// TwinCAT 3 PLC project Utilities
// Title: Tc_Utilities
// Company: NewEngineer
// Author: https://github.com/phucpha
// ProjectVersion: 1.1.1.0
// Description: this is library use for Utilities for TC3.
// ProgramVersion: 3.1.4024.0
// libraries:
//   Tc2_Standard, * (Beckhoff Automation GmbH)
//   Tc2_System, * (Beckhoff Automation GmbH)
//   Tc2_Utilities, * (Beckhoff Automation GmbH)
//   Tc3_Module, * (Beckhoff Automation GmbH)
// project tree:
//   DUTs/ E_3rdPartyScadaWriteDataBase.TcDUT
//   DUTs/File Logger/ E_FileLoggerAddLogsState.TcDUT (not stored), E_FileLoggerInitState.TcDUT (not stored), E_FileLoggerSetNewPathState.TcDUT (not stored), E_FileLoggerState.TcDUT (not stored)
//   DUTs/Union/ U_Word2Dint.TcDUT, U_Word2Int.TcDUT (not stored), U_Word2Real.TcDUT
//   FC/ FUN_Compare_Timestructs.TcPOU, TimeStruct_To_sTimeAveva.TcPOU
//   FC/StringMerge/ FUN_MergeLongStrings10.TcPOU, FUN_MergeStrings10.TcPOU, FUN_MergeStrings3.TcPOU, FUN_MergeStrings4.TcPOU (not stored), FUN_MergeStrings5.TcPOU, FUN_MergeStrings6.TcPOU
//   FC/Systemtime to String/ FUN_TimestructToDate.TcPOU, FUN_TimestructToTime.TcPOU
//   FC/ValueToTime/ F_lrMinute2Time.TcPOU, F_LrSecond2Time.TcPOU (not stored), F_Time2lrHour.TcPOU, F_Time2lrMinute.TcPOU (not stored), F_Time2lrSecond.TcPOU
//   GVLs/ GVL.TcGVL
//   / PlcTask.TcTTO
//   POUs/0_Checks/Checks/ CheckBounds.TcPOU, CheckDivDInt.TcPOU, CheckDivLInt.TcPOU, CheckDivLReal.TcPOU, CheckDivReal.TcPOU, CheckPointer.TcPOU, CheckRangeSigned.TcPOU, CheckRangeUnsigned.TcPOU, P_Checks.TcPOU
//   POUs/0_Checks/ GVL_Checks.TcGVL
//   POUs/Alarms/ FB_Alarm.TcPOU, I_Alarm.TcIO
//   POUs/CrossCheckTime/ FB_TimeCrossCheck2System.TcPOU
//   POUs/FileLogger/ FB_FileLogger.TcPOU (not stored), I_FileLogger.TcIO (not stored)
//   Version/ Global_Version.TcGVL
// real-time tasks:
//   TASK PlcTask: cycle T#10ms, priority 20, ADS port 350

CONFIGURATION Utilities
    RESOURCE PLC ON TwinCAT3
        TASK PlcTask(INTERVAL := T#10ms, PRIORITY := 20);
    END_RESOURCE
END_CONFIGURATION

// ---- DUTs/E_3rdPartyScadaWriteDataBase.TcDUT
{attribute 'strict'}
TYPE E_3rdPartyScadaWriteDataBase :
(
	DATABASE_WRITE_WAIT_START := 0,
	DATABASE_WRITE_PREPARE_VALUE, 
	DATABASE_WRITE_SEND_REQUEST,
	DATABASE_WRITE_WAIT_RESPONSE
	
);
END_TYPE

// ---- DUTs/Union/U_Word2Dint.TcDUT
TYPE U_Word2Dint :
UNION
	iWord	: ARRAY[0..1] OF WORD;
	idInt	: DINT;
END_UNION
END_TYPE

// ---- DUTs/Union/U_Word2Real.TcDUT
TYPE U_Word2Real :
UNION
	iWord: ARRAY [0..1] OF WORD;
	rReal: REAL;
END_UNION
END_TYPE

// ---- GVLs/GVL.TcGVL
VAR_GLOBAL
	fbMachineTime : FB_LocalSystemTime;
	fbMachineLogger : FB_FileLogger;
END_VAR

// ---- POUs/0_Checks/GVL_Checks.TcGVL
{attribute 'qualified_only'}
VAR_GLOBAL PERSISTENT
	dCheckBounds					: DINT;			// Licznik przekroczen zakresu indexow, np. tablic
	dCheckDivDInt					: DINT;			// Licznik prob dzielenia Dint przez 0
	dCheckDivLInt					: DINT; 		// Licznik prob dzielenia LInt przez 0
	dCheckDivLReal					: DINT; 		// Licznik prob dzielenia LREAL przez 0
	dCheckDivReal					: DINT; 		// Licznik prob dzielenia REAL przez 0
	dCheckRangeSigned				: DINT;			// Licznik przekroczen liczby znakowej
	dCheckRangeUnsigned				: DINT; 		// Licznik przekroczen liczby bezznakowej
END_VAR

// ---- Version/Global_Version.TcGVL
{attribute 'TcGenerated'}
{attribute 'no-analysis'}
{attribute 'linkalways'}
// This function has been automatically generated from the project information.
VAR_GLOBAL CONSTANT
	{attribute 'const_non_replaced'}
	stLibVersion_Tc_Utilities : ST_LibVersion := (iMajor := 1, iMinor := 1, iBuild := 1, iRevision := 0, nFlags := 0, sVersion := '1.1.1.0');
END_VAR

// ---- POUs/Alarms/I_Alarm.TcIO
INTERFACE I_Alarm

PROPERTY AlarmNumber : UINT
GET
END_GET
SET
END_SET
END_PROPERTY

PROPERTY Description : String
GET
END_GET
SET
END_SET
END_PROPERTY

METHOD Get : BOOL
VAR_INPUT
END_VAR
VAR_OUTPUT

END_VAR
END_METHOD

METHOD Reset : BOOL
VAR_INPUT
END_VAR
END_METHOD

METHOD Set : BOOL
VAR
END_VAR
VAR_INPUT
	bIn	:	BOOL;
END_VAR
END_METHOD

PROPERTY TimeOfOccur : TIMESTRUCT
GET
END_GET
END_PROPERTY

END_INTERFACE

// ---- FC/FUN_Compare_Timestructs.TcPOU
FUNCTION FUN_Compare_Timestructs : SINT //returns: 1 IF ts1 is older, -1 if ts2 is older, 0 if equal
VAR_INPUT
	ts1	:	TIMESTRUCT;
	ts2	:	TIMESTRUCT;
END_VAR
VAR
END_VAR

//OUTPUT: 1 IF ts1 is older, -1 if ts2 is older, 0 if equal
IF (ts1.wYear=ts2.wYear) THEN
	IF (ts1.wMonth=ts2.wMonth) THEN
		IF (ts1.wDay=ts2.wDay) THEN
			IF (ts1.wHour=ts2.wHour) THEN
				IF (ts1.wMinute=ts2.wMinute) THEN
					IF (ts1.wSecond=ts2.wSecond) THEN
						IF (ts1.wMilliseconds=ts2.wMilliseconds) THEN
							FUN_Compare_Timestructs:=0;
						ELSIF (ts1.wMilliseconds>ts2.wMilliseconds) THEN
								FUN_Compare_Timestructs:=-1;
						ELSE
								FUN_Compare_Timestructs:=1;
						END_IF
						
					ELSIF (ts1.wSecond>ts2.wSecond) THEN
						FUN_Compare_Timestructs:=-1;
					ELSE
						FUN_Compare_Timestructs:=1;
					END_IF
					
				ELSIF (ts1.wMinute>ts2.wMinute) THEN
					FUN_Compare_Timestructs:=-1;
				ELSE
					FUN_Compare_Timestructs:=1;
				END_IF
				
			ELSIF (ts1.wHour>ts2.wHour) THEN
				FUN_Compare_Timestructs:=-1;
			ELSE
				FUN_Compare_Timestructs:=1;
			END_IF
		
		ELSIF (ts1.wDay>ts2.wDay) THEN
			FUN_Compare_Timestructs:=-1;
		ELSE
			FUN_Compare_Timestructs:=1;
		END_IF
	
	ELSIF (ts1.wMonth>ts2.wMonth) THEN
		FUN_Compare_Timestructs:=-1;
	ELSE
		FUN_Compare_Timestructs:=1;
	END_IF
	
ELSIF (ts1.wYear>ts2.wYear) THEN
	FUN_Compare_Timestructs:=-1;
ELSE
	FUN_Compare_Timestructs:=1;
END_IF

END_FUNCTION

// ---- FC/StringMerge/FUN_MergeLongStrings10.TcPOU
(* 
:Description: This function is used to merge 10 long strings
*)
FUNCTION FUN_MergeLongStrings10 : STRING(2000)
VAR_INPUT
	sStr1	: STRING(2000);
	sStr2	: STRING(2000);
	sStr3	: STRING(2000);
	sStr4	: STRING(2000);
	sStr5	: STRING(2000);
	sStr6	: STRING(2000);
	sStr7	: STRING(2000);
	sStr8	: STRING(2000);
	sStr9	: STRING(2000);
	sStr10	: STRING(2000);
END_VAR
VAR
	sStrTemp1 :	STRING(2000);
	sStrTemp2 :	STRING(2000);
END_VAR

CONCAT2(ADR(sStr1),ADR(sStr2),ADR(sStrTemp1),SIZEOF(sStrTemp1));
CONCAT2(ADR(sStrTemp1),ADR(sStr3),ADR(sStrTemp2),SIZEOF(sStrTemp2));
CONCAT2(ADR(sStrTemp2),ADR(sStr4),ADR(sStrTemp1),SIZEOF(sStrTemp1));
CONCAT2(ADR(sStrTemp1),ADR(sStr5),ADR(sStrTemp2),SIZEOF(sStrTemp2));
CONCAT2(ADR(sStrTemp2),ADR(sStr6),ADR(sStrTemp1),SIZEOF(sStrTemp1));
CONCAT2(ADR(sStrTemp1),ADR(sStr7),ADR(sStrTemp2),SIZEOF(sStrTemp2));
CONCAT2(ADR(sStrTemp2),ADR(sStr8),ADR(sStrTemp1),SIZEOF(sStrTemp1));
CONCAT2(ADR(sStrTemp1),ADR(sStr9),ADR(sStrTemp2),SIZEOF(sStrTemp2));
CONCAT2(ADR(sStrTemp2),ADR(sStr10),ADR(FUN_MergeLongStrings10),SIZEOF(FUN_MergeLongStrings10));

END_FUNCTION

// ---- FC/StringMerge/FUN_MergeStrings10.TcPOU
(* 
:Description: This function is used to merge 10 strings
*)
FUNCTION FUN_MergeStrings10 : STRING
VAR_INPUT
	sStr1	: STRING;		(* First string in merge row *)
	sStr2	: STRING;		(* Second string in merge row *)
	sStr3	: STRING;		(* Third string in merge row *)
	sStr4	: STRING(500);	(* Fourth string in merge row *)
	sStr5	: STRING(500);	(* Fifth string in merge row *)
	sStr6	: STRING(500);	(* Sixth string in merge row *)
	sStr7	: STRING(500);	(* Seventh string in merge row *)
	sStr8	: STRING;		(* Eight string in merge row *)
	sStr9	: STRING;		(* Ninth string in merge row *)
	sStr10	: STRING;		(* Tenth string in merge row *)
END_VAR

FUN_MergeStrings10 := CONCAT(sStr1,sStr2);
FUN_MergeStrings10 := CONCAT(FUN_MergeStrings10,sStr3);
FUN_MergeStrings10 := CONCAT(FUN_MergeStrings10,sStr4);
FUN_MergeStrings10 := CONCAT(FUN_MergeStrings10,sStr5);
FUN_MergeStrings10 := CONCAT(FUN_MergeStrings10,sStr6);
FUN_MergeStrings10 := CONCAT(FUN_MergeStrings10,sStr7);
FUN_MergeStrings10 := CONCAT(FUN_MergeStrings10,sStr8);
FUN_MergeStrings10 := CONCAT(FUN_MergeStrings10,sStr9);
FUN_MergeStrings10 := CONCAT(FUN_MergeStrings10,sStr10);

END_FUNCTION

// ---- FC/StringMerge/FUN_MergeStrings3.TcPOU
(* 
:Description: This function is used to merge 5 strings
*)
FUNCTION FUN_MergeStrings3 : STRING
VAR_INPUT
	sStr1	: STRING;			(* Fifth string in merge row *)
	sStr2	: STRING;			(* Fourth string in merge row *)
	sStr3	: STRING;			(* Fourth string in merge row *)

END_VAR

FUN_MergeStrings3 := CONCAT(sStr1,sStr2);
FUN_MergeStrings3 := CONCAT(FUN_MergeStrings3,sStr3);

END_FUNCTION

// ---- FC/StringMerge/FUN_MergeStrings5.TcPOU
(* 
:Description: This function is used to merge 5 strings
*)
FUNCTION FUN_MergeStrings5 : STRING
VAR_INPUT
	sStr1	: STRING;		(* First string in merge row *)
	sStr2	: STRING;		(* Second string in merge row *)
	sStr3	: STRING;		(* Third string in merge row *)
	sStr4	: STRING;		(* Fourth string in merge row *)
	sStr5	: STRING;		(* Fifth string in merge row *)

END_VAR

FUN_MergeStrings5 := CONCAT(sStr1,sStr2);
FUN_MergeStrings5 := CONCAT(FUN_MergeStrings5, sStr3);
FUN_MergeStrings5 := CONCAT(FUN_MergeStrings5, sStr4);
FUN_MergeStrings5 := CONCAT(FUN_MergeStrings5, sStr5);

END_FUNCTION

// ---- FC/StringMerge/FUN_MergeStrings6.TcPOU
(* 
:Description: This function is used to merge 6 strings
*)
FUNCTION FUN_MergeStrings6 : STRING(300)
VAR_INPUT
	sStr1	: STRING;		(* First string in merge row *)
	sStr2	: STRING;		(* Second string in merge row *)
	sStr3	: STRING;		(* Third string in merge row *)
	sStr4	: STRING;		(* Fourth string in merge row *)
	sStr5	: STRING;		(* Fifth string in merge row *)
	sStr6	: STRING;		(* Sixth string in merge row *)
END_VAR

FUN_MergeStrings6 := CONCAT(sStr1,sStr2);
FUN_MergeStrings6 := CONCAT(FUN_MergeStrings6, sStr3);
FUN_MergeStrings6 := CONCAT(FUN_MergeStrings6, sStr4);
FUN_MergeStrings6 := CONCAT(FUN_MergeStrings6, sStr5);
FUN_MergeStrings6 := CONCAT(FUN_MergeStrings6, sStr6);

END_FUNCTION

// ---- FC/Systemtime to String/FUN_TimestructToDate.TcPOU
FUNCTION FUN_TimestructToDate : STRING
VAR_INPUT
	stTime : TIMESTRUCT;
END_VAR
VAR
	sTime : STRING;
END_VAR

sTime := SYSTEMTIME_TO_STRING(stTime);
FUN_TimestructToDate := LEFT(sTime,10);

END_FUNCTION

// ---- FC/Systemtime to String/FUN_TimestructToTime.TcPOU
FUNCTION FUN_TimestructToTime : STRING
VAR_INPUT
	stTime : TIMESTRUCT;
END_VAR
VAR
	sTime : STRING;
END_VAR

sTime := SYSTEMTIME_TO_STRING(stTime);
FUN_TimestructToTime := RIGHT(sTime,12);

END_FUNCTION

// ---- FC/TimeStruct_To_sTimeAveva.TcPOU
FUNCTION TimeStruct_To_sTimeAveva : STRING// convert TIMESTRUCT TO MONTH/DAY/YEAR HOUR:MINUTE: SECOND ( FORMAT 'MM/DD/YYYY HH:MM:SS' )
VAR_INPUT
	timestruct 	: TIMESTRUCT;
	typeFormat	: UINT := 0; (* 	0: 'MM/DD/YYYY HH:MM:SS'
									1: 'MMDDYYYY'
									2: 'YYYYMMDD'
									3: 'DDMMYYYY'
									4: 'YYYY-MM-DD HH:MM:SS' 
									5: 'YYYY-MM-DD HH:MM:SS.XXX'
													*)
	
END_VAR
VAR
	sYear : STRING;
	sMonth : STRING;
	sDay : STRING;
	sHour : STRING;
	sMinute : STRING;
	sSecond : STRING;
	sMilisecond	: STRING;
	concate1 : STRING;
	
END_VAR

	sYear := WORD_TO_STRING(timestruct.wYear);
	sMonth := WORD_TO_STRING(timestruct.wMonth);
	sDay 	:= WORD_TO_STRING(timestruct.wDay);
	
	sHour := WORD_TO_STRING(timestruct.wHour);
	sMinute := WORD_TO_STRING(timestruct.wMinute);
	sSecond 	:= WORD_TO_STRING(timestruct.wSecond);
	sMilisecond := WORD_TO_STRING(timestruct.wMilliseconds);
	
	IF timestruct.wMonth <10 THEN
		sMonth := CONCAT('0', smonth);
	END_IF
	
	IF timestruct.wDay <10 THEN
		sDay := CONCAT('0', sday);
	END_IF
	
	IF timestruct.wHour <10 THEN
		sHour := CONCAT('0', shour);
	END_IF
	IF timestruct.wSecond <10 THEN
		ssecond := CONCAT('0', ssecond);
	END_IF
	IF timestruct.wMinute <10 THEN
		sMinute := CONCAT('0', sminute);
	END_IF
	
	IF timestruct.wMilliseconds < 10  THEN
		sMilisecond :=  CONCAT('00', sMilisecond);
	ELSIF timestruct.wMilliseconds < 100 THEN
		sMilisecond :=  CONCAT('0', sMilisecond);
	END_IF
	
CASE typeFormat OF
	0://0: 'MM/DD/YYYY HH:MM:SS'
		concate1 := CONCAT( smonth, '/');
		concate1 := CONCAT( concate1, sDay);
		concate1 := CONCAT( concate1, '/');
		concate1 := CONCAT( concate1, sYear);
		concate1 := CONCAT( concate1, ' ');
		concate1 := CONCAT( concate1, shour);
		concate1 := CONCAT( concate1, ':');
		concate1 := CONCAT( concate1, sminute);
		concate1 := CONCAT( concate1, ':');
		concate1 := CONCAT( concate1, ssecond);
	
	1: //1: 'MMDDYYYY'
		concate1 := CONCAT( smonth, sDay);
		concate1 := CONCAT( concate1, sYear);
		
	2: 	//2: 'YYYYMMDD'
		concate1 := CONCAT( syear, smonth);
		concate1 := CONCAT( concate1, sday);	
		
	3: 	//3: 'DDMMYYYY'
		concate1 := CONCAT( sday, smonth);
		concate1 := CONCAT( concate1, syear);	
	4: //'YYYY-MM-DD HH:MM:SS' 
		concate1 := CONCAT( syear, '-');//YYYY-
		concate1 := CONCAT ( concate1, smonth);//YYYY-MM
		concate1 := CONCAT( concate1, '-');//YYYY-MM-
		concate1 := CONCAT( concate1, SDAY);//YYYY-MM-DD
		concate1 := CONCAT( concate1, ' ');//'YYYY-MM-DD '
		concate1 := CONCAT( concate1, shour);//'YYYY-MM-DD HH
		concate1 := CONCAT( concate1, ':');//'YYYY-MM-DD HH:
		concate1 := CONCAT( concate1, sminute);//'YYYY-MM-DD HH:MM
		concate1 := CONCAT( concate1, ':');//'YYYY-MM-DD HH:MM:
		concate1 := CONCAT( concate1, ssecond);//'YYYY-MM-DD HH:MM:SS
	5: (*need addition code*)
		concate1 := CONCAT( syear, '-');//YYYY-
		concate1 := CONCAT ( concate1, smonth);//YYYY-MM
		concate1 := CONCAT( concate1, '-');//YYYY-MM-
		concate1 := CONCAT( concate1, SDAY);//YYYY-MM-DD
		concate1 := CONCAT( concate1, ' ');//'YYYY-MM-DD '
		concate1 := CONCAT( concate1, shour);//'YYYY-MM-DD HH
		concate1 := CONCAT( concate1, ':');//'YYYY-MM-DD HH:
		concate1 := CONCAT( concate1, sminute);//'YYYY-MM-DD HH:MM
		concate1 := CONCAT( concate1, ':');//'YYYY-MM-DD HH:MM:
		concate1 := CONCAT( concate1, ssecond);//'YYYY-MM-DD HH:MM:SS
		concate1 := CONCAT( concate1, '.');//'YYYY-MM-DD HH:MM:SS.
		concate1 := CONCAT( concate1, sMilisecond); ////'YYYY-MM-DD HH:MM:SS.xxx
		
	ELSE
		concate1 := '';
END_CASE

TimeStruct_To_sTimeAveva := concate1;

END_FUNCTION

// ---- FC/ValueToTime/F_lrMinute2Time.TcPOU
FUNCTION F_lrMinute2Time : Time
VAR_INPUT
	lrMinute	: lreal;
END_VAR
VAR
END_VAR

F_lrMinute2Time := LREAL_TO_TIME( lrMinute*60*1000);

END_FUNCTION

// ---- FC/ValueToTime/F_Time2lrHour.TcPOU
FUNCTION F_Time2lrHour : lreal
VAR_INPUT
	t : TIME;
END_VAR

VAR
END_VAR

F_Time2lrHour := time_to_lreal(t)*2.777777777777777*expt(10,-7); // *0.001*0.01666666667 = /1000/60/60

END_FUNCTION

// ---- FC/ValueToTime/F_Time2lrSecond.TcPOU
FUNCTION F_Time2lrSecond : lreal
VAR_INPUT
	t : TIME;
END_VAR
VAR
END_VAR

F_Time2lrSecond := time_to_lreal(t)/1000;

END_FUNCTION

// ---- POUs/0_Checks/Checks/CheckBounds.TcPOU
// Implicitly generated code : DO NOT EDIT
FUNCTION CheckBounds : DINT
VAR_INPUT
	index, lower, upper: DINT;
END_VAR

// Implicitly generated code : Only an Implementation suggestion
IF  index < lower THEN
	CheckBounds := lower;
	GVL_Checks.dCheckBounds := GVL_Checks.dCheckBounds + 1;
//	ADSLOGSTR(4,'Checks critical error - index out of range','');
ELSIF  index > upper THEN
	CheckBounds := upper;
	GVL_Checks.dCheckBounds := GVL_Checks.dCheckBounds + 1;
//	ADSLOGSTR(4,'Checks critical error - index out of range','');
ELSE  
	CheckBounds := index;
END_IF

END_FUNCTION

// ---- POUs/0_Checks/Checks/CheckDivDInt.TcPOU
// Implicitly generated code : DO NOT EDIT
FUNCTION CheckDivDInt : DINT
VAR_INPUT
	divisor:DINT;
END_VAR

// Implicitly generated code : Only an Implementation suggestion
IF divisor = 0 THEN
	CheckDivDInt:=1;
	GVL_Checks.dCheckDivDInt := GVL_Checks.dCheckDivDInt + 1;
	ADSLOGSTR(4,'Checks critical error - DINT variable divided by 0.','');
ELSE
	CheckDivDInt:=divisor;
END_IF

END_FUNCTION

// ---- POUs/0_Checks/Checks/CheckDivLInt.TcPOU
// Implicitly generated code : DO NOT EDIT
FUNCTION CheckDivLInt : LINT
VAR_INPUT
	divisor:LINT;
END_VAR

// Implicitly generated code : Only an Implementation suggestion
IF divisor = 0 THEN
	CheckDivLInt:=1;
	GVL_Checks.dCheckDivLInt := GVL_Checks.dCheckDivLInt + 1;
	ADSLOGSTR(4,'Checks critical error - LINT variable divided by 0.','');
ELSE
	CheckDivLInt:=divisor;
END_IF

END_FUNCTION

// ---- POUs/0_Checks/Checks/CheckDivLReal.TcPOU
// Implicitly generated code : DO NOT EDIT
FUNCTION CheckDivLReal : LREAL
VAR_INPUT
	divisor:LREAL;
END_VAR

// Implicitly generated code : Only an Implementation suggestion
IF divisor = 0 THEN
	CheckDivLReal:=1;
	GVL_Checks.dCheckDivLReal := GVL_Checks.dCheckDivLReal + 1;
	ADSLOGSTR(4,'Checks critical error - DINT variable divided by 0.','');
ELSE
	CheckDivLReal:=divisor;
END_IF

END_FUNCTION

// ---- POUs/0_Checks/Checks/CheckDivReal.TcPOU
// Implicitly generated code : DO NOT EDIT
FUNCTION CheckDivReal : REAL
VAR_INPUT
	divisor:REAL;
END_VAR

// Implicitly generated code : Only an Implementation suggestion
IF divisor = 0 THEN
	CheckDivReal:=1;
	GVL_Checks.dCheckDivReal := GVL_Checks.dCheckDivReal + 1;
	ADSLOGSTR(4,'Checks critical error - DINT variable divided by 0.','');
ELSE
	CheckDivReal:=divisor;
END_IF

END_FUNCTION

// ---- POUs/0_Checks/Checks/CheckPointer.TcPOU
// Implicitly generated code : DO NOT EDIT
FUNCTION CheckPointer : POINTER TO BYTE
VAR_INPUT 
	ptToTest : POINTER TO BYTE; // Destination address of the pointer
	iSize : DINT;		        // Size of the type the pointer points to. (e.g: 20 for POINTER TO ARRAY [0..9] OF INT) 
	iGran : DINT;		        // Granularity of the pointer access. This is the size of the biggest non-structured data type in the type the pointer points to. (e.g: 2 for POINTER TO ARRAY [0..9] OF INT)
	bWrite: BOOL;		        // Indicates read or write Access. TRUE = write access.
END_VAR

// No standard way of implementation. Fill your own code here
CheckPointer := ptToTest;

END_FUNCTION

// ---- POUs/0_Checks/Checks/CheckRangeSigned.TcPOU
// Implicitly generated code : DO NOT EDIT
FUNCTION CheckRangeSigned : DINT
VAR_INPUT
	value, lower, upper: DINT;
END_VAR

// Implicitly generated code : Only an Implementation suggestion
IF (value < lower) THEN
	CheckRangeSigned := lower;
	GVL_Checks.dCheckRangeSigned := GVL_Checks.dCheckRangeSigned + 1;
	ADSLOGSTR(4,'Checks critical error - DINT overflow.','');
ELSIF(value > upper) THEN
	CheckRangeSigned := upper;
	GVL_Checks.dCheckRangeSigned := GVL_Checks.dCheckRangeSigned + 1;
	ADSLOGSTR(4,'Checks critical error - DINT overflow.','');
ELSE
	CheckRangeSigned := value;
END_IF

END_FUNCTION

// ---- POUs/0_Checks/Checks/CheckRangeUnsigned.TcPOU
// Implicitly generated code : DO NOT EDIT
FUNCTION CheckRangeUnsigned : UDINT
VAR_INPUT
	value, lower, upper: UDINT;
END_VAR

// Implicitly generated code : Only an Implementation suggestion
IF (value < lower) THEN
	CheckRangeUnsigned := lower;
	GVL_Checks.dCheckRangeUnsigned := GVL_Checks.dCheckRangeUnsigned + 1;
	ADSLOGSTR(4,'Checks critical error - UDINT overflow.','');
ELSIF(value > upper) THEN
	CheckRangeUnsigned := upper;
	GVL_Checks.dCheckRangeUnsigned := GVL_Checks.dCheckRangeUnsigned + 1;
	ADSLOGSTR(4,'Checks critical error - UDINT overflow.','');
ELSE
	CheckRangeUnsigned := value;
END_IF

END_FUNCTION

// ---- POUs/0_Checks/Checks/P_Checks.TcPOU
PROGRAM P_Checks
VAR_INPUT
	bReset							: BOOL;
END_VAR
VAR_OUTPUT
	bOK								: BOOL;	// Brak bledow i ostrzezen
	bWarning						: BOOL;	// Ostrzezenie - nie wystepuja w tym podprogramie - wystepuja dla zachowania spojnosci
	bError							: BOOL;	// Zbiorcza flaga bledow
END_VAR
VAR
	bCheckBounds					: BOOL;	// Flaga przekroczen zakresu indexow, np. tablic
	bCheckDivDInt					: BOOL;	// Flaga prob dzielenia Dint przez 0
	bCheckDivLInt					: BOOL; // Flaga prob dzielenia LInt przez 0
	bCheckDivLReal					: BOOL; // Flaga prob dzielenia LREAL przez 0
	bCheckDivReal					: BOOL; // Flaga prob dzielenia REAL przez 0
	bCheckRangeSigned				: BOOL;	// Flaga przekroczen liczby znakowej
	bCheckRangeUnsigned				: BOOL; // Flaga przekroczen liczby bezznakowej
	
	dCheckBoundsOld					: DINT;	// Licznik przekroczen zakresu indexow, np. tablic
	dCheckDivDIntOld				: DINT;	// Licznik prob dzielenia Dint przez 0
	dCheckDivLIntOld				: DINT; // Licznik prob dzielenia LInt przez 0
	dCheckDivLRealOld				: DINT; // Licznik prob dzielenia LREAL przez 0
	dCheckDivRealOld				: DINT; // Licznik prob dzielenia REAL przez 0
	dCheckRangeSignedOld			: DINT;	// Licznik przekroczen  liczby znakowej
	dCheckRangeUnsignedOld			: DINT; // Licznik przekroczen  liczby bezznakowej
END_VAR

IF bReset THEN
	bCheckBounds 					:= FALSE;
	bCheckDivDInt					:= FALSE;
	bCheckDivLInt					:= FALSE;
	bCheckDivLReal					:= FALSE;
	bCheckDivReal					:= FALSE;
	bCheckRangeSigned				:= FALSE;
	bCheckRangeUnsigned				:= FALSE;
ELSE
	bCheckBounds 					S= dCheckBoundsOld <> GVL_Checks.dCheckBounds;
	bCheckDivDInt					S= dCheckDivDIntOld <> GVL_Checks.dCheckDivDInt;
	bCheckDivLInt					S= dCheckDivLIntOld <> GVL_Checks.dCheckDivLInt;
	bCheckDivLReal					S= dCheckDivLRealOld <> GVL_Checks.dCheckDivLReal;
	bCheckDivReal					S= dCheckDivRealOld <> GVL_Checks.dCheckDivReal;
	bCheckRangeSigned				S= dCheckRangeSignedOld <> GVL_Checks.dCheckRangeSigned;
	bCheckRangeUnsigned				S= dCheckRangeUnsignedOld <> GVL_Checks.dCheckRangeUnsigned;	
END_IF

dCheckBoundsOld 					:= GVL_Checks.dCheckBounds;
dCheckDivDIntOld 					:= GVL_Checks.dCheckDivDInt;
dCheckDivLIntOld 					:= GVL_Checks.dCheckDivLInt;
dCheckDivLRealOld 					:= GVL_Checks.dCheckDivLReal;
dCheckDivRealOld 					:= GVL_Checks.dCheckDivReal;
dCheckRangeSignedOld 				:= GVL_Checks.dCheckRangeSigned;
dCheckRangeUnsignedOld 				:= GVL_Checks.dCheckRangeUnsigned;

bError 								:= bCheckBounds OR bCheckDivDInt OR bCheckDivLInt OR bCheckDivLReal OR bCheckDivReal OR bCheckRangeSigned OR bCheckRangeUnsigned;
bOK 								:= NOT bError AND NOT bWarning;

END_PROGRAM

// ---- POUs/Alarms/FB_Alarm.TcPOU
FUNCTION_BLOCK FB_Alarm IMPLEMENTS I_Alarm
VAR_INPUT
END_VAR
VAR_OUTPUT
END_VAR
VAR
	iAlarmNumber	:	UINT := 0;
	bTemporary		:	BOOL;
	bLatched		:	BOOL;
	sDescription	:	STRING;
	tsTimeOfOccur	:	TIMESTRUCT;
END_VAR

{attribute 'monitoring' := 'variable'}
PROPERTY AlarmNumber : UINT
GET
AlarmNumber := iAlarmNumber;
END_GET
SET
iAlarmNumber := AlarmNumber;
END_SET
END_PROPERTY

{attribute 'monitoring' := 'variable'}
PROPERTY Description : String
GET
Description := sDescription;
END_GET
SET
sDescription := Description;
END_SET
END_PROPERTY

METHOD Get : BOOL
VAR_INPUT
END_VAR
VAR_OUTPUT

END_VAR
Get := bLatched;
END_METHOD

METHOD Reset : BOOL
VAR_INPUT
END_VAR
IF NOT bTemporary THEN
	IF bLatched = TRUE THEN
		Reset := TRUE;
		bLatched := FALSE;
	END_IF
ELSE
	Reset := FALSE;
END_IF
END_METHOD

METHOD Set : BOOL
VAR
END_VAR
VAR_INPUT
	bIn	:	BOOL;
END_VAR
bTemporary := bIn;
IF NOT bLatched AND bIn THEN
	bLatched := TRUE;
	tsTimeOfOccur := GVL.fbMachineTime.systemTime;
END_IF
END_METHOD

PROPERTY TimeOfOccur : TIMESTRUCT
GET
TimeOfOccur := tsTimeOfOccur;
END_GET
END_PROPERTY

END_FUNCTION_BLOCK

// ---- POUs/CrossCheckTime/FB_TimeCrossCheck2System.TcPOU
FUNCTION_BLOCK FB_TimeCrossCheck2System
VAR_INPUT
	TimeStruct_Sys1 : TIMESTRUCT;
 	TimeStruct_Sys2 : TIMESTRUCT;
	secondDifferentAllow : UDINT; 
END_VAR
VAR_OUTPUT
	bErrorTimeTwoSystem : BOOL;
END_VAR
VAR
	DtSys1 : DT;
	DtSys2 : DT;
	uDSys1 : LREAL;
	uDsys2 : LREAL;
	diferent : lreal;
	
END_VAR


DtSys1 := SYSTEMTIME_TO_DT(TimeStruct_Sys1);
DtSys2 := SYSTEMTIME_TO_DT(TimeStruct_Sys2);

uDSys1 := DT_TO_LREAL(DtSys1);
uDSys2 := DT_TO_LREAL(DtSys2);
diferent := uDSys1 - uDsys2;
IF ABS(uDSys1 - uDsys2) > secondDifferentAllow THEN
	bErrorTimeTwoSystem := TRUE;
ELSE
	bErrorTimeTwoSystem := FALSE;
END_IF

END_FUNCTION_BLOCK
